// TIA Portal V20 export
DATA_BLOCK "DB_Vacuums"   // DB441
// stored: AutoNumber false, InstanceOfName FB_Vacuums, InstanceOfType FB
"FB_Vacuums"
   // VAR
   //    sOutVacuum1On : Bool;
   //    sControlVacuum1 { S7_SetPoint := 'True'} : "FB_AnalogInputThreshold";
   //    sCtrlPressureVacuum1 { S7_SetPoint := 'True'} : "FB_AnalogInputThreshold";
   //    sAspirationLeft { S7_SetPoint := 'True'} : "FB_AnalogInputThreshold";
   //    sAspirationRight { S7_SetPoint := 'True'} : "FB_AnalogInputThreshold";
   //    sRT_AspirationKeys { S7_SetPoint := 'True'} : R_TRIG;
   //    sFT_AspirationKeys { S7_SetPoint := 'True'} : F_TRIG;
   //    sAspirationKeys { S7_SetPoint := 'True'} : Bool;
   // END_VAR
BEGIN
END_DATA_BLOCK
